// TIA Portal V19 export
TYPE "C103_VAR_IF_OVI_TYPIC"
   STRUCT
      SCL { ExternalAccessible := 'False'; ExternalVisible := 'False'; ExternalWritable := 'False'} : Bool;   // Standmelding aankomstschakelaar
   END_STRUCT;
END_TYPE
